// TwinCAT 3 PLC project array_fun
// ProgramVersion: 3.1.4024.0
// libraries:
//   Tc2_Standard, * (Beckhoff Automation GmbH)
//   Tc2_System, * (Beckhoff Automation GmbH)
//   Tc3_Module, * (Beckhoff Automation GmbH)
// project tree:
//   DUTs/ MyStructure.TcDUT
//   / PlcTask.TcTTO
//   POUs/ FB_RollerDoor.TcPOU, GVL_Doors.TcGVL, MAIN.TcPOU, RollerDoors.TcPOU, sRollerDoor.TcDUT
// real-time tasks:
//   TASK PlcTask: cycle T#10ms, priority 20, ADS port 350

CONFIGURATION array_fun
    RESOURCE PLC ON TwinCAT3
        TASK PlcTask(INTERVAL := T#10ms, PRIORITY := 20);
        PROGRAM MAIN WITH PlcTask : MAIN;
    END_RESOURCE
END_CONFIGURATION

// ---- DUTs/MyStructure.TcDUT
TYPE MyStructure :
STRUCT
	Var1 : INT;    // Serial number (will change)
    Var2 : REAL;   // Constant value
    Var3 : BOOL;   // Constant value
    Var4 : TIME;   // Constant time value
    Var5 : STRING[20]; // Constant string value
END_STRUCT
END_TYPE

// ---- POUs/sRollerDoor.TcDUT
TYPE sRollerDoor :
STRUCT
	ManualOpenRequest	: BOOL;
	ManualCloseRequest	: BOOL;
	AutoOpenRequest	 	: BOOL;
	AutoCloseRequest	: BOOL;
		
	CommandOpenOutput	AT %Q* : BOOL;		
	CommandCloseOutput	AT %Q* : BOOL;
	
	StatusOpenedInput	AT %I* : BOOL; //This is Normally Closed
	StatusClosedInput	AT %I* : BOOL; //This is Normally Closed
	
	// DOOR_OPEN_SWITCH AT %I*: BOOL;// REAL WORLD SWITCH INPUT
	// DOOR_CLOSED_SWITCH AT %I*: BOOL; // REAL WORLD SWITCH INPUT
	DOOR_CLEAR AT %I* : BOOL; // LIGHT CURTAIN CLEAR
	// RUN_UP AT %Q* : BOOL; // DISCRETE OUTPUT FOR RAISE DOOR COMMAND
	// RUN_DOWN AT %Q* : BOOL; // DISCRETE OUTPUT FOR LOWER DOOR COMMAND
	DOOR_OPEN:BOOL; // DOOR CURRENT POSITION IS OPEN
	DOOR_CLOSED:BOOL; // DOOR CURRENT POSITION IS CLOSED
	OPEN_REQUEST:BOOL; // PLC REQUESTING ROLL DOOR TO OPEN
	CLOSE_REQUEST:BOOL; // PLC REQUESTING ROLL DOOR TO CLOSE
	UP_SWITCH_IS_ON:BOOL; // DOOR SWITCH FOR UP POSITION IS ON
	UP_SWITCH_IS_OFF:BOOL; // DOOR SWITCH FOR UP POSITION IS OFF
	DOWN_SWITCH_IS_ON:BOOL; // DOOR SWITCH FOR DOWN POSITION IS ON
	DOWN_SWITCH_IS_OFF:BOOL; // DOOR SWITCH FOR DOWN POSITION IS OFF
	
	
	DOOR_IS_UP_TimerOn : TON;
	DOOR_IS_UP_TimerOn_Done_Bit: BOOL;
	DOOR_IS_UP_TIMER_ON_ELAPSED : TIME;
	
	DOOR_IS_UP_TimerOFF : TOF;
	DOOR_IS_UP_TimerOFF_Done_Bit: BOOL;
	DOOR_IS_UP_TIMER_OFF_ELAPSED : TIME;
	
	DOOR_IS_DOWN_TimerOn : TON;
	DOOR_IS_DOWN_TimerOn_Done_Bit: BOOL;
	DOOR_IS_DOWN_TIMER_ON_ELAPSED : TIME;
	
	DOOR_IS_DOWN_TimerOFF : TOF;
	DOOR_IS_DOWN_TimerOFF_Done_Bit: BOOL;
	DOOR_IS_DOWN_TIMER_OFF_ELAPSED : TIME;
	
END_STRUCT
END_TYPE

// ---- POUs/GVL_Doors.TcGVL
rahu{attribute 'qualified_only'}
VAR_GLOBAL
	FQ1 : sRollerDoor;	//Smaller Roller Door - Input to Spray Zone at GL5B
	FQ2 : sRollerDoor;	//Larger Roller Door on SD1
	FQ3 : sRollerDoor;	//Larger Roller Door on SD2
	RibDoor: sRollerDoor; // Door to process enclosure to pass ribs through to pick and place
	QQ1 : sPersonnelDoor; //Sliding Personnel Door
	FQ4	: sRollerDoor;	// Front porch roll up door at GL12
END_VAR

// ---- POUs/MAIN.TcPOU
PROGRAM MAIN
VAR
MyArray : ARRAY[1..100] OF MyStructure;  // Array of 100 structures
    i : INT;  // Loop index
	binputbools AT %I*:ARRAY [1..4] OF BOOL;
	boutputbools AT %Q*:ARRAY [1..4]OF BOOL;
	d:BOOL;
	h:int;
	
END_VAR




FOR i := 1 TO 100 DO
    MyArray[i].Var1 := i;             // Assign serial number 1 to 100 to Var1
    MyArray[i].Var2 := 105.9;          // Set constant value for Var2
    MyArray[i].Var3 := TRUE;          // Set constant value for Var3
    MyArray[i].Var4 := T#1s;          // Set constant time value for Var4
    MyArray[i].Var5 := 'Serial #' ;  // Set a unique string for each structure
END_FOR

END_PROGRAM

// ---- POUs/FB_RollerDoor.TcPOU
FUNCTION_BLOCK FB_RollerDoor
VAR_INPUT
	AutoMode : BOOL;
	ManualMode : BOOL;
	ManualDoorOpenRequest : BOOL;
	ManualDoorCloseRequest : BOOL;
	AutoDoorOpenRequest : BOOL;
	AutoDoorCloseRequest : BOOL;
	StatusOpenedInput : BOOL;
	StatusClosedInput : BOOL;
	test:BOOL;
	
	
END_VAR
VAR_OUTPUT
	DoorOpenCommand : BOOL;
	DoorCloseCommand : BOOL;
END_VAR
VAR
	ManualDoorOpenRequestRTRIG : R_TRIG;
	ManualDoorCloseRequestRTRIG : R_TRIG;
	AutoDoorOpenRequestRTRIG : R_TRIG;
	AutoDoorCloseRequestRTRIG : R_TRIG;
END_VAR

IF AutoMode THEN
	
	AutoDoorOpenRequestRTRIG(CLK := AutoDoorOpenRequest);
	AutoDoorCloseRequestRTRIG(CLK := AutoDoorCloseRequest);
	
	IF AutoDoorOpenRequestRTRIG.Q THEN
		DoorOpenCommand := 1;
		DoorCloseCommand := 0;
	ELSIF AutoDoorCloseRequestRTRIG.Q THEN
		DoorCloseCommand := 1;
		DoorOpenCommand := 0;
	END_IF
	IF StatusOpenedInput THEN 
		DoorOpenCommand := 0;
	END_IF

	IF StatusClosedInput THEN 
		DoorCloseCommand := 0;
	END_IF
	
END_IF

IF ManualMode THEN
	
	ManualDoorOpenRequestRTRIG(CLK := ManualDoorOpenRequest);
	ManualDoorCloseRequestRTRIG(CLK := ManualDoorCloseRequest);
	
	IF ManualDoorOpenRequestRTRIG.Q THEN
		DoorOpenCommand := 1;
		DoorCloseCommand := 0;
	ELSIF ManualDoorCloseRequestRTRIG.Q THEN
		DoorCloseCommand := 1;
		DoorOpenCommand := 0;
	END_IF
END_IF

END_FUNCTION_BLOCK

// ---- POUs/RollerDoors.TcPOU
PROGRAM RollerDoors
VAR
	FQ1_FB : FB_RollerDoor;
	FQ2_FB : FB_RollerDoor;
	FQ3_FB : FB_RollerDoor;
	FQ4_FB : FB_RollerDoor;
	
END_VAR

//The Bogies control FQ2 and FQ3 on SD1 and SD2, respectively. 
//the conveyors are controlling all other doors

//FQ1 shuttle Roller Door
IF GVL_Doors.FQ1.StatusOpenedInput THEN 
	GVL_Doors.FQ1.AutoOpenRequest := 0;
	GVL_Doors.FQ1.CommandOpenOutput := FALSE;
END_IF

IF GVL_Doors.FQ1.StatusClosedInput THEN 
	GVL_Doors.FQ1.AutoCloseRequest := 0;
	GVL_Doors.FQ1.CommandCloseOutput := FALSE;
END_IF

FQ1_FB(	AutoMode				:= GVL_HMI.AutoMode,
		ManualMode 				:= GVL_HMI.ManualMode,
		ManualDoorOpenRequest	:= GVL_Doors.FQ1.ManualOpenRequest,
		ManualDoorCloseRequest 	:= GVL_Doors.FQ1.ManualCloseRequest,
		AutoDoorOpenRequest 	:= GVL_Doors.FQ1.AutoOpenRequest,
		AutoDoorCloseRequest 	:= GVL_Doors.FQ1.AutoCloseRequest,
		DoorOpenCommand 		=> GVL_Doors.FQ1.CommandOpenOutput,
		DoorCloseCommand 		=> GVL_Doors.FQ1.CommandCloseOutput,
		StatusOpenedInput		:= GVL_Doors.FQ1.StatusOpenedInput,
		StatusClosedInput		:= GVL_Doors.FQ1.StatusClosedInput);
		
GVL_Doors.FQ1.CommandOpenOutput		:= FQ1_FB.DoorOpenCommand;
GVL_Doors.FQ1.CommandCloseOutput	:= FQ1_FB.DoorCloseCommand;
FQ1_FB();



//FQ2 SD1 Roller Door
IF GVL_Doors.FQ2.StatusOpenedInput THEN 
	GVL_Doors.FQ2.AutoOpenRequest := 0;
	GVL_Doors.FQ2.CommandOpenOutput := FALSE;
END_IF

IF GVL_Doors.FQ2.StatusClosedInput THEN 
	GVL_Doors.FQ2.AutoCloseRequest := 0;
	GVL_Doors.FQ2.CommandCloseOutput := FALSE;
END_IF

FQ2_FB(	AutoMode				:= GVL_HMI.AutoMode,
		ManualMode 				:= GVL_HMI.ManualMode,
		ManualDoorOpenRequest	:= GVL_Doors.FQ2.ManualOpenRequest,
		ManualDoorCloseRequest 	:= GVL_Doors.FQ2.ManualCloseRequest,
		AutoDoorOpenRequest 	:= GVL_Doors.FQ2.AutoOpenRequest,
		AutoDoorCloseRequest 	:= GVL_Doors.FQ2.AutoCloseRequest,
		DoorOpenCommand 		=> GVL_Doors.FQ2.CommandOpenOutput,
		DoorCloseCommand 		=> GVL_Doors.FQ2.CommandCloseOutput,
		StatusOpenedInput		:= GVL_Doors.FQ2.StatusOpenedInput,
		StatusClosedInput		:= GVL_Doors.FQ2.StatusClosedInput);
		
GVL_Doors.FQ2.CommandOpenOutput		:= FQ2_FB.DoorOpenCommand;
GVL_Doors.FQ2.CommandCloseOutput	:= FQ2_FB.DoorCloseCommand;
FQ2_FB(); // Update function block to reset outputs

//FQ3 SD2 Roller Door
IF GVL_Doors.FQ3.StatusOpenedInput THEN 
	GVL_Doors.FQ3.AutoOpenRequest := 0;
	GVL_Doors.FQ3.CommandOpenOutput := FALSE;
END_IF

IF GVL_Doors.FQ3.StatusClosedInput THEN 
	GVL_Doors.FQ3.AutoCloseRequest := 0;
	GVL_Doors.FQ3.CommandCloseOutput := FALSE;
END_IF
		
FQ3_FB(	AutoMode				:= GVL_HMI.AutoMode,
		ManualMode 				:= GVL_HMI.ManualMode,
		ManualDoorOpenRequest	:= GVL_Doors.FQ3.ManualOpenRequest,
		ManualDoorCloseRequest 	:= GVL_Doors.FQ3.ManualCloseRequest,
		AutoDoorOpenRequest 	:= GVL_Doors.FQ3.AutoOpenRequest,
		AutoDoorCloseRequest 	:= GVL_Doors.FQ3.AutoCloseRequest,
		DoorOpenCommand 		=> GVL_Doors.FQ3.CommandOpenOutput,
		DoorCloseCommand 		=> GVL_Doors.FQ3.CommandCloseOutput,
		StatusOpenedInput		:= GVL_Doors.FQ3.StatusOpenedInput,
		StatusClosedInput		:= GVL_Doors.FQ3.StatusClosedInput
		);

GVL_Doors.FQ3.CommandOpenOutput		:= FQ3_FB.DoorOpenCommand;
GVL_Doors.FQ3.CommandCloseOutput	:= FQ3_FB.DoorCloseCommand;
FQ3_FB(); // Update function block to reset outputs
	

//FQ4 GL12 Roller Door
IF GVL_Doors.FQ4.StatusOpenedInput THEN 
	GVL_Doors.FQ4.AutoOpenRequest := 0;
	GVL_Doors.FQ4.CommandOpenOutput := FALSE;
END_IF

IF GVL_Doors.FQ4.StatusClosedInput THEN 
	GVL_Doors.FQ4.AutoCloseRequest := 0;
	GVL_Doors.FQ4.CommandCloseOutput := FALSE;
END_IF
		
FQ4_FB(	AutoMode				:= GVL_HMI.AutoMode,
		ManualMode 				:= GVL_HMI.ManualMode,
		ManualDoorOpenRequest	:= GVL_Doors.FQ4.ManualOpenRequest,
		ManualDoorCloseRequest 	:= GVL_Doors.FQ4.ManualCloseRequest,
		AutoDoorOpenRequest 	:= GVL_Doors.FQ4.AutoOpenRequest,
		AutoDoorCloseRequest 	:= GVL_Doors.FQ4.AutoCloseRequest,
		DoorOpenCommand 		=> GVL_Doors.FQ4.CommandOpenOutput,
		DoorCloseCommand 		=> GVL_Doors.FQ4.CommandCloseOutput,
		StatusOpenedInput		:= GVL_Doors.FQ3.StatusOpenedInput,
		StatusClosedInput		:= GVL_Doors.FQ3.StatusClosedInput);

GVL_Doors.FQ4.CommandOpenOutput		:= FQ4_FB.DoorOpenCommand;
GVL_Doors.FQ4.CommandCloseOutput	:= FQ4_FB.DoorCloseCommand;

FQ4_FB(); // Update function block to reset outputs

END_PROGRAM
